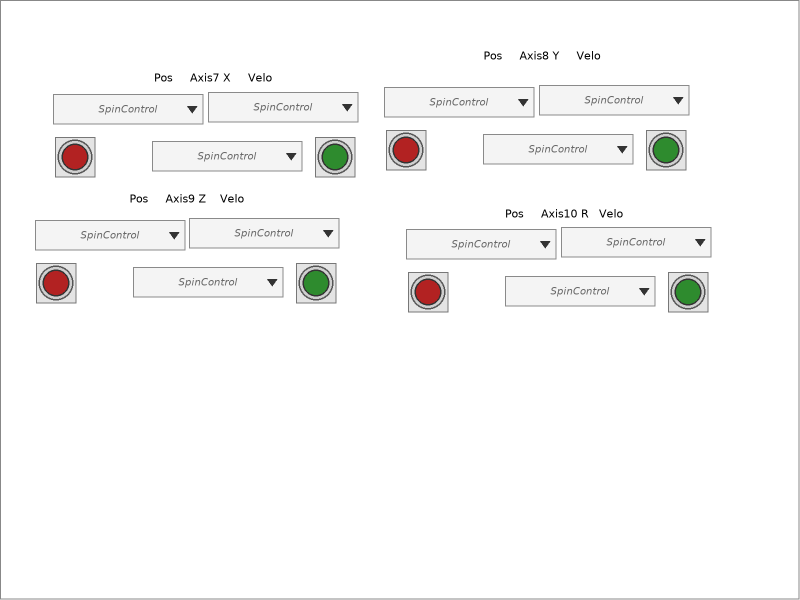
VISUALIZATION ManiMotors  // 800x600
    SpinControl (406,229 150x30), variable: Axis10.rPosition
    PushSwitch (408,272 40x40), variable: Axis10.boHalt, behaviour: TOGGLE, style: Switch-PushSwitch-Red
    PushSwitch (668,272 40x40), variable: Axis10.boMoveAbsolute, behaviour: TOGGLE, style: Switch-PushSwitch-Green
    SpinControl (505,276 150x30), variable: Axis10.roPosition
    SpinControl (561,227 150x30), variable: Axis10.rVelocity
    Label (489,199 150x30), "Pos Axis10 R Velo"
    PushSwitch (36,263 40x40), variable: Axis9.boHalt, behaviour: TOGGLE, style: Switch-PushSwitch-Red
    SpinControl (35,220 150x30), variable: Axis9.rPosition
    PushSwitch (296,263 40x40), variable: Axis9.boMoveAbsolute, behaviour: TOGGLE, style: Switch-PushSwitch-Green
    SpinControl (133,267 150x30), variable: Axis9.roPosition
        p1653691745: 0.05
    SpinControl (189,218 150x30), variable: Axis9.rVelocity
    PushSwitch (386,130 40x40), variable: Axis8.boHalt, behaviour: TOGGLE, style: Switch-PushSwitch-Red
    SpinControl (384,87 150x30), variable: Axis8.rPosition
    PushSwitch (646,130 40x40), variable: Axis8.boMoveAbsolute, behaviour: TOGGLE, style: Switch-PushSwitch-Green
    SpinControl (483,134 150x30), variable: Axis8.roPosition
        p1653691745: 0.05
    SpinControl (539,85 150x30), variable: Axis8.rVelocity
    PushSwitch (55,137 40x40), variable: Axis7.boHalt, behaviour: TOGGLE, style: Switch-PushSwitch-Red
    SpinControl (53,94 150x30), variable: Axis7.rPosition
    PushSwitch (315,137 40x40), variable: Axis7.boMoveAbsolute, behaviour: TOGGLE, style: Switch-PushSwitch-Green
    SpinControl (152,141 150x30), variable: Axis7.roPosition
        p1653691745: 0.05
    SpinControl (208,92 150x30), variable: Axis7.rVelocity
    Label (112,184 150x30), "Pos Axis9 Z Velo"
    Label (467,41 150x30), "Pos Axis8 Y Velo"
    Label (138,63 150x30), "Pos Axis7 X Velo"
END_VISUALIZATION

(* stored: Version 1.1.0.1, ProductVersion 3.1.4022.3
   Visu ManiMotors: Id {272a3e35-2ff1-4c23-94e1-593f70d427ab} *)
